INTERFACE I_JobNode EXTENDS I_JobNodeInternal

END_INTERFACE

(* stored: Version 1.1.0.1
   Itf I_JobNode: Id {d740f790-ee67-445b-9a56-dbf77aaa8b7e} *)
